{attribute 'linkalways'} 
{attribute 'no_explicit_call' := 'This FB is a CLASS and must be accessed using methods or properties'}
{attribute 'enable_dynamic_creation'}
FUNCTION_BLOCK Node_F_VN_SubtractVectorFromImage EXTENDS VisionNode
VAR
    ipSrcImage : _ITcVnImage;
    aVector : _TcVnVector4_LREAL;
    ipDestImage : _ITcVnImage;
    hrPrev : _HRESULT(S_OK);
	hresult : _HRESULT(S_OK);
END_VAR

METHOD PUBLIC  Clone : I_Node
VAR
	pNode : POINTER TO Node_F_VN_SubtractVectorFromImage;
END_VAR
pNode := __NEW(Node_F_VN_SubtractVectorFromImage);
Clone := pNode^;
END_METHOD

METHOD FB_init : BOOL
VAR_INPUT
	bInitRetains : BOOL; // if TRUE, the retain variables are initialized (warm start / cold start)
	bInCopyCode : BOOL;  // if TRUE, the instance afterwards gets moved into the copy code (online change)
END_VAR
AddInput('ipSrcImage', ipSrcImage);
AddInput('aVector', aVector);
AddInput('hrPrev', hrPrev);
AddOutput('ipDestImage', ipDestImage);
AddOutput('hresult',hresult);
END_METHOD

METHOD PROTECTED OnExecute
hresult.Value := F_VN_SubtractVectorFromImage(
    ipSrcImage := ipSrcImage.Value,
    aVector := aVector.Value,
	ipDestImage := ipDestImage.Value,
	hrPrev:= hrPrev.Value);
END_METHOD

METHOD PUBLIC PreExecutionCheck
VAR_INPUT
	Check : I_PreExecutionChecks;
END_VAR
Check.IsTrue(ipSrcImage.IsValid, 'ipSrcImage must contain an image');
END_METHOD

END_FUNCTION_BLOCK

(* stored: Version 1.1.0.1, ProductVersion 3.1.4024.13
   POU Node_F_VN_SubtractVectorFromImage: Id {bb92132f-a06f-0583-24d6-ca8f121932fe}, SpecialFunc None
   Folder Constructor: Id {93894e47-6303-022e-322f-9b11a109de12}
   Method Clone: Id {08c2a371-230b-0ebc-12c1-f71471eb66e7}
   Method FB_init: Id {92e73927-85a2-0a62-2bc9-95900487ac9d}
   Method OnExecute: Id {b1f6037d-591a-047b-360a-9ced0879a25c}
   Method PreExecutionCheck: Id {c99c4913-ccb5-0b57-0413-6986f050ec56} *)
